Staubli VAL3: ActiviteEleve.dtx

pointRs pp1 = {x=6.500000, y=219.500000, z=15.500000, rx=-180, ry=-5.500000e-15, rz=-55.000000, fatherId=world[0]}
pointRs pp2 = {x=20.500000, y=219.000000, z=92.500000, rx=-180, ry=-5.500000e-15, rz=-55.000000, fatherId=world[0]}
pointRs pp3 = {x=-18.500000, y=-219.000000, z=80.000000, rx=180, ry=5.500000e-15, rz=125.500000, fatherId=world[0]}
pointRs pp4 = {x=-9.500000, y=-219.000000, z=7.000000, rx=180, ry=5.500000e-15, rz=123.000000, fatherId=world[0]}
